PROGRAM MAIN
VAR
END_VAR

END_PROGRAM

(* stored: Version 1.1.0.1
   POU MAIN: Id {ef8c1139-ee97-43ae-bca4-6c0b7c990c6b} *)
